TYPE ActuatorConfiguration EXTENDS BaseConfiguration:
STRUCT
	//Output
	sPusherType : STRING;
	iPusherPosition : DINT;
END_STRUCT
END_TYPE

(* stored: Version 1.1.0.1
   DUT ActuatorConfiguration: Id {1df0ba73-301f-48a2-a571-27e7b4736ffc} *)
